FUNCTION_BLOCK ILOCK_CONFLICT_TRIP_PROTECT_AX (* Prioritizes the first active input and trips on conflict, with protection dead-time after release (Adapter Version). Requires RESET. *)
  (* Standard: 61499-2; Description: Copyright (c) 2026 Meisterschulen am Ostbahnhof This program and the accompanying materials are made available under the terms of the Eclipse Public License 2.0 which is available at https://www.eclipse.org/legal/epl-2.0/ SPDX-License-Identifier: EPL-2.0 *)
  (* Version 1.0, 2026-09-07, Franz Höpfinger, Meisterschulen am Ostbahnhof, ILOCK_CONFLICT_TRIP_AX + Totzeit nach Freigabe (UPDATE/DT_PROTECT/timeOut wie ILOCK_BLOCK_PROTECT_AX) - TRAINING_GAPS.md Punkt 6 *)
  PACKAGE logiBUS::signalprocessing::interlock;
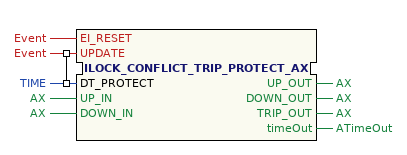
  EVENT_INPUT
    EI_RESET;
    UPDATE WITH DT_PROTECT; (* Update parameters *)
  END_EVENT
  VAR_INPUT
    DT_PROTECT : TIME := T#50ms; (* Protection Time *)
  END_VAR
  SOCKETS
    UP_IN : adapter::types::unidirectional::AX; (* Input for forward/up direction *)
    DOWN_IN : adapter::types::unidirectional::AX; (* Input for backward/down direction *)
  END_SOCKETS
  PLUGS
    UP_OUT : adapter::types::unidirectional::AX; (* Output for forward/up direction *)
    DOWN_OUT : adapter::types::unidirectional::AX; (* Output for backward/down direction *)
    TRIP_OUT : adapter::types::unidirectional::AX; (* Trip State Output *)
    timeOut : iec61499::events::ATimeOut; (* timeOut Adapter *)
  END_PLUGS
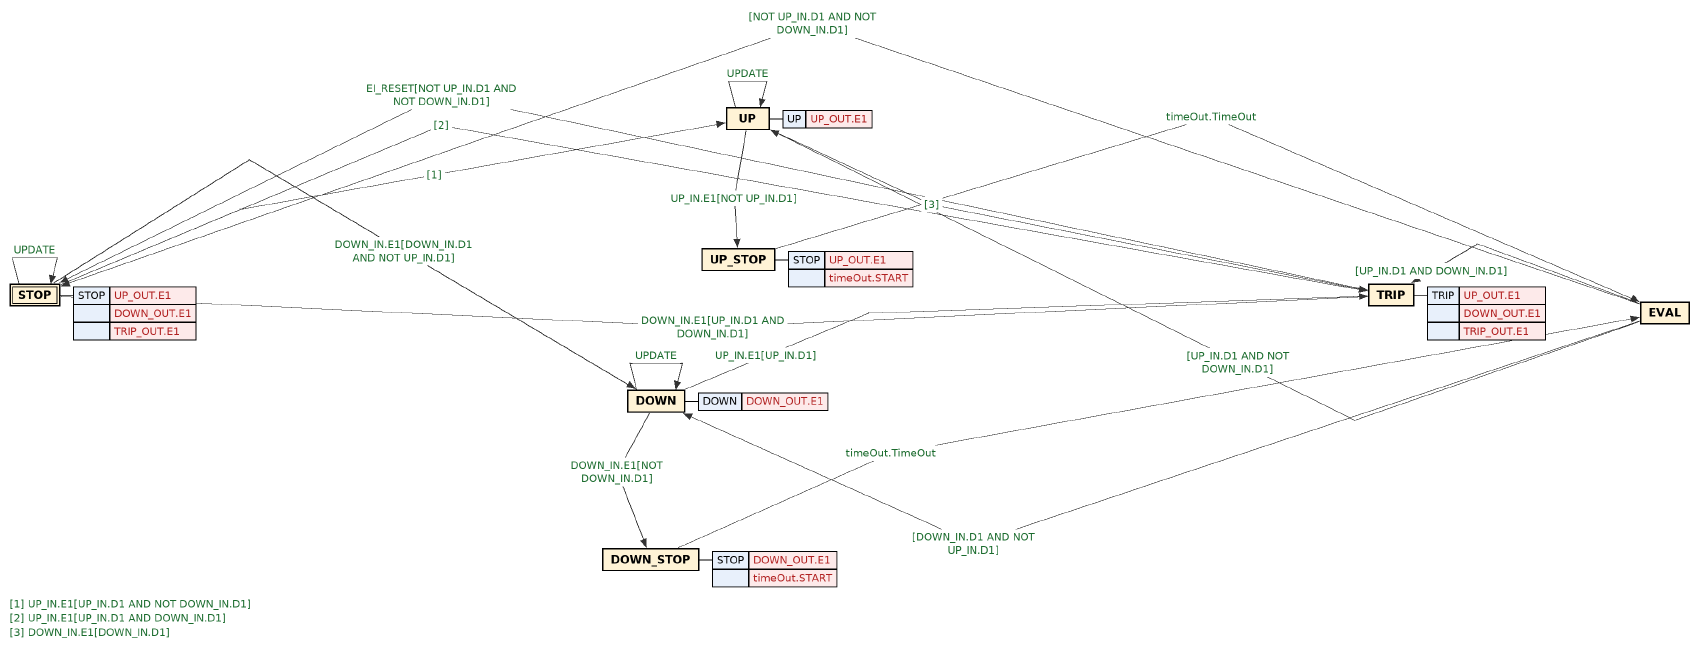
  EC_STATES
    STOP : STOP -> UP_OUT.E1, -> DOWN_OUT.E1, -> TRIP_OUT.E1;
    UP : UP -> UP_OUT.E1;
    DOWN : DOWN -> DOWN_OUT.E1;
    TRIP : TRIP -> UP_OUT.E1, -> DOWN_OUT.E1, -> TRIP_OUT.E1;
    UP_STOP : STOP -> UP_OUT.E1, -> timeOut.START;
    DOWN_STOP : STOP -> DOWN_OUT.E1, -> timeOut.START;
    EVAL;
  END_STATES
  EC_TRANSITIONS
    STOP TO UP := UP_IN.E1[UP_IN.D1 AND NOT DOWN_IN.D1];
    STOP TO DOWN := DOWN_IN.E1[DOWN_IN.D1 AND NOT UP_IN.D1];
    STOP TO TRIP := UP_IN.E1[UP_IN.D1 AND DOWN_IN.D1];
    STOP TO TRIP := DOWN_IN.E1[UP_IN.D1 AND DOWN_IN.D1];
    UP TO UP_STOP := UP_IN.E1[NOT UP_IN.D1];
    UP TO TRIP := DOWN_IN.E1[DOWN_IN.D1];
    DOWN TO DOWN_STOP := DOWN_IN.E1[NOT DOWN_IN.D1];
    DOWN TO TRIP := UP_IN.E1[UP_IN.D1];
    UP_STOP TO EVAL := timeOut.TimeOut;
    DOWN_STOP TO EVAL := timeOut.TimeOut;
    EVAL TO UP := [UP_IN.D1 AND NOT DOWN_IN.D1];
    EVAL TO DOWN := [DOWN_IN.D1 AND NOT UP_IN.D1];
    EVAL TO STOP := [NOT UP_IN.D1 AND NOT DOWN_IN.D1];
    EVAL TO TRIP := [UP_IN.D1 AND DOWN_IN.D1];
    TRIP TO STOP := EI_RESET[NOT UP_IN.D1 AND NOT DOWN_IN.D1];
    STOP TO STOP := UPDATE;
    UP TO UP := UPDATE;
    DOWN TO DOWN := UPDATE;
  END_TRANSITIONS
  ALGORITHM UP IN ST:
timeOut.DT := DT_PROTECT;
UP_OUT.D1 := BOOL#TRUE;
DOWN_OUT.D1 := BOOL#FALSE;
TRIP_OUT.D1 := BOOL#FALSE;
  END_ALGORITHM
  ALGORITHM DOWN IN ST:
timeOut.DT := DT_PROTECT;
UP_OUT.D1 := BOOL#FALSE;
DOWN_OUT.D1 := BOOL#TRUE;
TRIP_OUT.D1 := BOOL#FALSE;
  END_ALGORITHM
  ALGORITHM STOP IN ST:
timeOut.DT := DT_PROTECT;
UP_OUT.D1 := BOOL#FALSE;
DOWN_OUT.D1 := BOOL#FALSE;
TRIP_OUT.D1 := BOOL#FALSE;
  END_ALGORITHM
  ALGORITHM TRIP IN ST:
UP_OUT.D1 := BOOL#FALSE;
DOWN_OUT.D1 := BOOL#FALSE;
TRIP_OUT.D1 := BOOL#TRUE;
  END_ALGORITHM
END_FUNCTION_BLOCK
